INTERFACE I_Jog EXTENDS I_Axis

METHOD Inch : HRESULT
VAR_INPUT
	Distance : MC_LREAL;
	Direction : BOOL;
END_VAR
END_METHOD

METHOD JogFast : HRESULT
VAR_INPUT
	Direction : BOOL;
END_VAR
END_METHOD

METHOD JogSlow : HRESULT
VAR_INPUT
	Direction : BOOL;
END_VAR
END_METHOD

END_INTERFACE

(* stored: Version 1.1.0.1
   Itf I_Jog: Id {8e49aba1-c725-4b7a-a4e0-47b9b3e8e5b3}
   Method Inch: Id {281576ff-057a-4763-8087-52cdeebb4e0f}
   Method JogFast: Id {5ccbd402-3762-490b-87e3-2aa40d5a5ec5}
   Method JogSlow: Id {4c6aefe1-eed0-4a63-b373-fddbc3ed5508} *)
